// TIA Portal V19 export
VAR_GLOBAL   // PLC tag table "Safety Tags"
   "ESTOP CH1" AT %I18.1 : Bool;
   Estop_LED AT %Q24.0 : Bool;
   "RFID_Gate CH1" AT %I18.0 : Bool;
   RFID_Gate_AUX AT %I22.2 : Bool;
   Safety_PB_Blue_Lamp AT %M90.0 : Bool;
END_VAR
